// TwinCAT 3 PLC project Base_Lib
// Title: Base Library
// Company: Beckhoff UK
// Author: Chris Knight
// ProjectVersion: 3.3.0
// ProgramVersion: 3.1.4026.25
// libraries:
//   Tc2_Standard, * (Beckhoff Automation GmbH)
//   Tc2_System, * (Beckhoff Automation GmbH)
//   Tc3_EventLogger, * (Beckhoff Automation GmbH)
// project tree:
//   Base Types/Abort_Base/ I_Abortable.TcIO
//   Base Types/Cyclic_Base/ CyclicBase.TcPOU, I_Cyclic.TcIO
//   Base Types/Initialise/ I_Initialisable.TcIO
//   Base Types/Object/ I_Object.TcIO, Object.TcPOU
//   Base Types/Reset_Base/ I_Resettable.TcIO
//   Base Types/Task_Base/ I_Task.TcIO, TaskBase.TcPOU, TaskExecutionStates.TcDUT
//   Cyclic Runner/ I_HostObjects.TcIO, I_RunObjects.TcIO, ObjectRunner.TcPOU
//   Project Information/ F_GetCompany.TcPOU, F_GetTitle.TcPOU, F_GetVersion.TcPOU
//   Tracing/ AdsLogger.TcPOU, EventLogger.TcPOU, I_Trace.TcIO, I_TraceLogger.TcIO, I_TracePublisher.TcIO, TcEventSeverityExt.TcDUT, Trace.TcPOU, Tracing.TcGVL
//   Version/ Global_Version.TcGVL

// ---- Base Types/Task_Base/TaskExecutionStates.TcDUT
{attribute 'qualified_only'}
{attribute 'strict'}
{attribute 'to_string'}
TYPE TaskExecutionStates :
(
	Idle := 0,
	Running := 1,
	Done := 2,
	Error := 3
);
END_TYPE

// ---- Tracing/TcEventSeverityExt.TcDUT
{attribute 'qualified_only'}
{attribute 'strict'}
{attribute 'to_string'}
TYPE TcEventSeverityExt : (
		Verbose	 := 0,
		Info	 := 1,
		Warning	 := 2,
		Error	 := 3,
		Critical := 4,
		Off		 := 5
	);
END_TYPE

// ---- Tracing/Tracing.TcGVL
{attribute 'qualified_only'}
VAR_GLOBAL
	Trace : Trace<10> := (TraceLevel := TcEventSeverityExt.Verbose);
	{attribute 'hide'}
	AdsLogger : AdsLogger(Trace);
	TcEventLogger : EventLogger(Trace);
END_VAR

// ---- Version/Global_Version.TcGVL
{attribute 'TcGenerated'}
{attribute 'no-analysis'}
{attribute 'linkalways'}
// This function has been automatically generated from the project information.
VAR_GLOBAL CONSTANT
	{attribute 'const_non_replaced'}
	stLibVersion_Base_Library : ST_LibVersion := (iMajor := 3, iMinor := 3, iBuild := 0, iRevision := 0, nFlags := 0, sVersion := '3.3.0');
END_VAR

// ---- Base Types/Abort_Base/I_Abortable.TcIO
INTERFACE I_Abortable EXTENDS __SYSTEM.IQueryInterface

METHOD Abort : HRESULT
VAR_INPUT
END_VAR
END_METHOD

END_INTERFACE

// ---- Base Types/Cyclic_Base/I_Cyclic.TcIO
INTERFACE I_Cyclic EXTENDS __SYSTEM.IQueryInterface

METHOD PUBLIC Cycle : HRESULT
VAR_INPUT
END_VAR
END_METHOD

END_INTERFACE

// ---- Base Types/Initialise/I_Initialisable.TcIO
INTERFACE I_Initialisable EXTENDS __SYSTEM.IQueryInterface

METHOD Initialise : HRESULT
VAR_INPUT
END_VAR
END_METHOD

PROPERTY Initialised : BOOL
GET
END_GET
END_PROPERTY

END_INTERFACE

// ---- Base Types/Object/I_Object.TcIO
INTERFACE I_Object

METHOD RegisterWithParent
VAR_INPUT
	Parent : I_HostObjects;
END_VAR
END_METHOD

END_INTERFACE

// ---- Base Types/Reset_Base/I_Resettable.TcIO
INTERFACE I_Resettable

METHOD PUBLIC Reset : HRESULT
VAR_INPUT
END_VAR
END_METHOD

END_INTERFACE

// ---- Base Types/Task_Base/I_Task.TcIO
INTERFACE I_Task EXTENDS I_Cyclic

PROPERTY Busy : bool
GET
END_GET
END_PROPERTY

PROPERTY Done : bool
GET
END_GET
END_PROPERTY

PROPERTY Error : bool
GET
END_GET
END_PROPERTY

END_INTERFACE

// ---- Cyclic Runner/I_HostObjects.TcIO
INTERFACE I_HostObjects

METHOD RegisterAbortable : HRESULT
VAR_INPUT
	Abortable : I_Abortable;
END_VAR
END_METHOD

METHOD RegisterCyclic : HRESULT
VAR_INPUT
	Cyclic : I_Cyclic;
END_VAR
END_METHOD

METHOD RegisterInitialisable : HRESULT
VAR_INPUT
	Initialisable : I_Initialisable;
END_VAR
END_METHOD

METHOD RegisterObject : HRESULT
VAR_INPUT
	Object : I_Object;
END_VAR
END_METHOD

METHOD RegisterResettable : HRESULT
VAR_INPUT
	Resetable : I_Resettable;
END_VAR
END_METHOD

METHOD RegisterTask : HRESULT
VAR_INPUT
	Task : I_Task;
END_VAR
END_METHOD

END_INTERFACE

// ---- Cyclic Runner/I_RunObjects.TcIO
INTERFACE I_RunObjects

METHOD Abort : HRESULT
VAR_INPUT
END_VAR
END_METHOD

METHOD PUBLIC  Cycle : HRESULT
VAR_INPUT
END_VAR
END_METHOD

METHOD DeregisterAll : HRESULT
VAR_INPUT
END_VAR
END_METHOD

METHOD Initialise : HRESULT
END_METHOD

METHOD Initialise_Ordered : HRESULT
END_METHOD

METHOD Register : HRESULT
VAR_INPUT
	Registerable : I_Object;
END_VAR
END_METHOD

METHOD Reset : HRESULT
VAR_INPUT
END_VAR
END_METHOD

END_INTERFACE

// ---- Tracing/I_Trace.TcIO
INTERFACE I_Trace

METHOD Critical
VAR_INPUT
	Source	  : T_MaxString;
	Message	  : T_MaxString;
END_VAR
END_METHOD

METHOD Error
VAR_INPUT
	Source	  : T_MaxString;
	Message	  : T_MaxString;
END_VAR
END_METHOD

METHOD Info
VAR_INPUT
	Source	  : T_MaxString;
	Message	  : T_MaxString;
END_VAR
END_METHOD

METHOD Verbose
VAR_INPUT
	Source	  : T_MaxString;
	Message	  : T_MaxString;
END_VAR
END_METHOD

METHOD Warning
VAR_INPUT
	Source	  : T_MaxString;
	Message	  : T_MaxString;
END_VAR
END_METHOD

END_INTERFACE

// ---- Tracing/I_TraceLogger.TcIO
INTERFACE I_TraceLogger

METHOD LogMessage
VAR_INPUT
	Key		  : T_MaxString;
	Value	  : T_MaxString;
	SourceId  : UDINT := 0;
	TimeStamp : ULINT := 0;
	MessageId : UDINT := 1;
	Severity  : USINT := 1;
END_VAR
END_METHOD

END_INTERFACE

// ---- Tracing/I_TracePublisher.TcIO
INTERFACE I_TracePublisher

METHOD Subscribe
VAR_INPUT
	Logger : I_TraceLogger;
END_VAR
END_METHOD

METHOD Unsubscribe
VAR_INPUT
	Logger : I_TraceLogger;
END_VAR
END_METHOD

END_INTERFACE

// ---- Tracing/Trace.TcPOU
FUNCTION_BLOCK Trace
VAR_GENERIC CONSTANT
	MaxCount : UDINT := 10;
END_VAR IMPLEMENTS I_TracePublisher, I_Trace
VAR
	Loggers : ARRAY[0..MaxCount] OF I_TraceLogger;
	_TraceLevel : TcEventSeverityExt := TcEventSeverityExt.Warning;
END_VAR

METHOD Critical
VAR_INPUT
	Source	  : T_MaxString;
	Message	  : T_MaxString;
END_VAR
VAR
	i : UDINT;
END_VAR
FOR i := 0 TO MaxCount DO
	IF Loggers[i] <> 0 AND_THEN _TraceLevel < 5 THEN
		Loggers[i].LogMessage(Source,
							  Message,
							  0,
							  0,
							  1,
							  4);
	END_IF
END_FOR
END_METHOD

METHOD Error
VAR_INPUT
	Source	  : T_MaxString;
	Message	  : T_MaxString;
END_VAR
VAR
	i : UDINT;
END_VAR
FOR i := 0 TO MaxCount DO
	IF Loggers[i] <> 0 AND_THEN _TraceLevel < 4 THEN
		Loggers[i].LogMessage(Source,
							  Message,
							  0,
							  0,
							  1,
							  3);
	END_IF
END_FOR
END_METHOD

METHOD Info
VAR_INPUT
	Source	  : T_MaxString;
	Message	  : T_MaxString;
END_VAR
VAR
	i : UDINT;
END_VAR
FOR i := 0 TO MaxCount DO
	IF Loggers[i] <> 0 AND_THEN _TraceLevel < 2 THEN
		Loggers[i].LogMessage(Source,
							  Message,
							  0,
							  0,
							  1,
							  1);
	END_IF
END_FOR
END_METHOD

METHOD Subscribe
VAR_INPUT
	Logger : I_TraceLogger;
END_VAR

VAR
	i : UDINT;
END_VAR
FOR i := 0 TO MaxCount DO
	IF Loggers[i] = 0 THEN
		Loggers[i] := Logger;
		EXIT;
	END_IF
END_FOR
END_METHOD

PROPERTY TraceLevel : TcEventSeverityExt
GET
TraceLevel := _TraceLevel;
END_GET
SET
_TraceLevel := TraceLevel;
END_SET
END_PROPERTY

METHOD Unsubscribe
VAR_INPUT
	Logger : I_TraceLogger;
END_VAR

VAR
	i : UDINT;
END_VAR
FOR i := 0 TO MaxCount DO
	IF Loggers[i] = Logger THEN
		Loggers[i] := 0;
		EXIT;
	END_IF
END_FOR
END_METHOD

METHOD Verbose
VAR_INPUT
	Source	  : T_MaxString;
	Message	  : T_MaxString;
END_VAR
VAR
	i : UDINT;
END_VAR
FOR i := 0 TO MaxCount DO
	IF Loggers[i] <> 0 AND_THEN _TraceLevel = 0 THEN
		Loggers[i].LogMessage(Source,
							  Message,
							  0,
							  0,
							  1,
							  0);
	END_IF
END_FOR
END_METHOD

METHOD Warning
VAR_INPUT
	Source	  : T_MaxString;
	Message	  : T_MaxString;
END_VAR
VAR
	i : UDINT;
END_VAR
FOR i := 0 TO MaxCount DO
	IF Loggers[i] <> 0 AND_THEN _TraceLevel < 3 THEN
		Loggers[i].LogMessage(Source,
							  Message,
							  0,
							  0,
							  1,
							  2);
	END_IF
END_FOR
END_METHOD

END_FUNCTION_BLOCK

// ---- Tracing/AdsLogger.TcPOU
FUNCTION_BLOCK AdsLogger IMPLEMENTS I_TraceLogger
VAR
	MessagesThisScan : DINT;
	CurrentCycle	 : UDINT;
END_VAR

//FB_Init is always available implicitly and it is used primarily for initialization.

//The return value is not evaluated. For a specific influence, you can also declare the

//methods explicitly and provide additional code there with the standard initialization

//code. You can evaluate the return value.
METHOD FB_Init : BOOL
VAR_INPUT
	bInitRetains   : BOOL; // TRUE: the retain variables are initialized (reset warm / reset cold)
	bInCopyCode	   : BOOL; // TRUE: the instance will be copied to the copy code afterward (online change)   
	TracePublisher : I_TracePublisher;
END_VAR
TracePublisher.Subscribe(THIS^);
END_METHOD

METHOD LogMessage
VAR_INPUT
	Key		  : T_MaxString;
	Value	  : T_MaxString;
	SourceId  : UDINT := 0;
	TimeStamp : ULINT := 0;
	MessageId : UDINT := 1;
	Severity  : USINT := 1;
END_VAR
IF TwinCAT_SystemInfoVarList._TaskInfo[GETCURTASKINDEXEX()].CycleCount <> CurrentCycle THEN
	CurrentCycle	 := TwinCAT_SystemInfoVarList._TaskInfo[GETCURTASKINDEXEX()].CycleCount;
	MessagesThisScan := 0;
END_IF

IF NOT (MessagesThisScan < TO_DINT(TwinCAT_SystemInfoVarList._TaskInfo[GETCURTASKINDEXEX()].CycleTime / 2000)) THEN
	RETURN;
END_IF

IF MessagesThisScan < TO_DINT(TwinCAT_SystemInfoVarList._TaskInfo[GETCURTASKINDEXEX()].CycleTime / 2000) THEN
	CASE Severity OF
		0,1:
			ADSLOGSTR(ADSLOG_MSGTYPE_LOG OR ADSLOG_MSGTYPE_HINT, Concat(Key, ': %s'), Value);
		2:
			ADSLOGSTR(ADSLOG_MSGTYPE_LOG OR ADSLOG_MSGTYPE_WARN, Concat(Key, ': %s'), Value);
		3,4:
			ADSLOGSTR(ADSLOG_MSGTYPE_LOG OR ADSLOG_MSGTYPE_ERROR, Concat(Key, ': %s'), Value);
	END_CASE
	
	MessagesThisScan := MessagesThisScan + 1;
END_IF
END_METHOD

END_FUNCTION_BLOCK

// ---- Tracing/EventLogger.TcPOU
FUNCTION_BLOCK EventLogger IMPLEMENTS I_TraceLogger
VAR
	MessagesThisScan : DINT;
	Message			 : FB_TcMessage;
	Source			 : FB_TcSourceInfo;
	CurrentCycle	 : UDINT;
END_VAR

//FB_Init is always available implicitly and it is used primarily for initialization.
//The return value is not evaluated. For a specific influence, you can also declare the
//methods explicitly and provide additional code there with the standard initialization
//code. You can evaluate the return value.
METHOD FB_Init: BOOL
VAR_INPUT
    bInitRetains: BOOL; // TRUE: the retain variables are initialized (reset warm / reset cold)
    bInCopyCode: BOOL;  // TRUE: the instance will be copied to the copy code afterward (online change)   
	TracePublisher : I_TracePublisher;	
END_VAR
TracePublisher.Subscribe(THIS^);
END_METHOD

METHOD LogMessage
VAR_INPUT
	Key	: T_MaxString;
	Value	: T_MaxString;
	SourceId	: UDINT := 0;
	TimeStamp	: ULINT := 0;
	MessageId	: UDINT := 1;
	Severity	: USINT := 1;
END_VAR
VAR
	EventSeverity : TcEventSeverity;
END_VAR
IF TwinCAT_SystemInfoVarList._TaskInfo[GETCURTASKINDEXEX()].CycleCount <> CurrentCycle THEN
	CurrentCycle	 := TwinCAT_SystemInfoVarList._TaskInfo[GETCURTASKINDEXEX()].CycleCount;
	MessagesThisScan := 0;
END_IF

IF NOT (MessagesThisScan < TO_DINT(TwinCAT_SystemInfoVarList._TaskInfo[GETCURTASKINDEXEX()].CycleTime / 2000)) THEN
	RETURN;
END_IF

CASE Severity OF
	0: 
		EventSeverity := TcEventSeverity.Verbose;

	1:
		EventSeverity := TcEventSeverity.Info;

	2:
		EventSeverity := TcEventSeverity.Warning;

	3:
		EventSeverity := TcEventSeverity.Error;

	4:
		EventSeverity := TcEventSeverity.Critical;
END_CASE

Source.sName := Key;
Source.nId	 := SourceId;
Message.Create(eventClass	:= TC_EVENT_CLASSES.TraceEvents,
			   nEventId		:= MessageId,
			   eSeverity	:= EventSeverity,
			   ipSourceInfo := Source);

Message.ipArguments.Clear().AddString(Value);
Message.Send(TimeStamp);
Message.Release();
Source.Clear();
MessagesThisScan := MessagesThisScan + 1;
END_METHOD

END_FUNCTION_BLOCK

// ---- Base Types/Cyclic_Base/CyclicBase.TcPOU
FUNCTION_BLOCK ABSTRACT CyclicBase EXTENDS Object IMPLEMENTS I_Cyclic
VAR
END_VAR

{analysis -2}

METHOD PUBLIC ABSTRACT Cycle : HRESULT
VAR_INPUT
END_VAR
{analysis -2}
END_METHOD

METHOD RegisterWithParent
VAR_INPUT
	Parent	: I_HostObjects;
END_VAR
Parent.RegisterObject(THIS^);
Parent.RegisterCyclic(THIS^);
END_METHOD

END_FUNCTION_BLOCK

// ---- Base Types/Object/Object.TcPOU
FUNCTION_BLOCK ABSTRACT Object IMPLEMENTS I_Object
VAR
	_Name : T_MaxString;
END_VAR

//FB_Init is always available implicitly and it is used primarily for initialization.
//The return value is not evaluated. For a specific influence, you can also declare the
//methods explicitly and provide additional code there with the standard initialization
//code. You can evaluate the return value.
METHOD FB_Init: BOOL
VAR_INPUT
    bInitRetains: BOOL; // TRUE: the retain variables are initialized (reset warm / reset cold)
    bInCopyCode: BOOL;  // TRUE: the instance will be copied to the copy code afterward (online change)  
	Name : T_MaxString; 
END_VAR
_Name := Name;
END_METHOD

PROPERTY Name : T_MaxString
GET
Name := _Name;
END_GET
END_PROPERTY

METHOD RegisterWithParent
VAR_INPUT
	Parent	: I_HostObjects;
END_VAR
Parent.RegisterObject(THIS^);
END_METHOD

END_FUNCTION_BLOCK

// ---- Base Types/Task_Base/TaskBase.TcPOU
FUNCTION_BLOCK ABSTRACT TaskBase EXTENDS CyclicBase IMPLEMENTS I_Task
VAR
	_Busy : BOOL;
	_Error : BOOL;
	_Done : BOOL;
	State: INT;
END_VAR

{analysis -2}

PROPERTY Busy : BOOL
GET
Busy := _Busy;
END_GET
END_PROPERTY

PROPERTY Done : BOOL
GET
Done := _Done;
END_GET
END_PROPERTY

PROPERTY Error : BOOL
GET
Error := _Error;
END_GET
END_PROPERTY

END_FUNCTION_BLOCK

// ---- Cyclic Runner/ObjectRunner.TcPOU
FUNCTION_BLOCK ObjectRunner 
VAR_GENERIC CONSTANT
	MaxRegisteredModules : INT := 99;
END_VAR IMPLEMENTS I_Cyclic, I_HostObjects, I_RunObjects
VAR
	Objects : ARRAY[0..MaxRegisteredModules] OF I_Object;
	CyclicModules : ARRAY[0..MaxRegisteredModules] OF I_Cyclic;
	InitialiseModules : ARRAY[0..MaxRegisteredModules] OF I_Initialisable;
	ResetableModules : ARRAY[0..MaxRegisteredModules] OF I_Resettable;
	AbortableModules : ARRAY[0..MaxRegisteredModules] OF I_Abortable;
	TaskModules : ARRAY[0..MaxRegisteredModules] OF I_Task;
	_ObjectCount : INT := 0;
	_CyclicModuleCount : INT := 0;
	_InitModuleCount : INT := 0;
	_ResetModuleCount : INT := 0;
	_TaskModuleCount : INT := 0;
	_AbortModuleCount: INT := 0;
	InitialisationCount : INT := 0;
	Registered: BOOL;
	_AllInitialised : BOOL := TRUE;
END_VAR

METHOD Abort : HRESULT
VAR_INPUT
END_VAR
VAR	
	i: INT;
END_VAR
IF _AbortModuleCount = 0 THEN
	Abort := -1;
	RETURN;
END_IF

FOR i := 0 TO _AbortModuleCount - 1 DO
	IF AbortableModules[i] <> 0 THEN
		AbortableModules[i].Abort();
	END_IF
END_FOR
END_METHOD

PROPERTY AbortableModuleCount : INT
GET
AbortableModuleCount := _AbortModuleCount;
END_GET
END_PROPERTY

METHOD PUBLIC  Cycle : HRESULT
VAR_INPUT
END_VAR
VAR	
	i: INT;
END_VAR
FOR i := 0 TO _CyclicModuleCount -1 DO
	IF CyclicModules[i] <> 0 THEN
		CyclicModules[i].Cycle();
	END_IF
END_FOR
END_METHOD

PROPERTY CyclicModuleCount : INT
GET
CyclicModuleCount := _CyclicModuleCount;
END_GET
END_PROPERTY

METHOD DeregisterAll : HRESULT
VAR_INPUT
END_VAR
VAR	
	i: INT;
END_VAR
FOR i := 0 TO MaxRegisteredModules DO
	Objects[i] := 0;
	CyclicModules[i] := 0;
	InitialiseModules[i] := 0;
	ResetableModules[i] := 0;
	AbortableModules[i] := 0;
	TaskModules[i] := 0;
END_FOR
_CyclicModuleCount := 0;
_InitModuleCount := 0;
_ResetModuleCount := 0;
_TaskModuleCount := 0;
_AbortModuleCount := 0;
InitialisationCount := 0;
_ObjectCount := 0;
DeregisterAll := 1;
END_METHOD

PROPERTY InitialisableModuleCount : INT
GET
InitialisableModuleCount := _InitModuleCount;
END_GET
END_PROPERTY

PROPERTY InitialisationComplete : BOOL
GET
InitialisationComplete := _AllInitialised;
END_GET
END_PROPERTY

METHOD Initialise : HRESULT
VAR
	i : INT;
END_VAR
IF _InitModuleCount = 0 THEN
	_AllInitialised := TRUE;
	RETURN; 
END_IF

_AllInitialised := TRUE;
FOR i := 0 TO _InitModuleCount DO
	IF InitialiseModules[i] <> 0 THEN 
		IF NOT InitialiseModules[i].Initialised THEN
			InitialiseModules[i].Initialise();
			_AllInitialised := FALSE;
			Initialise := -1;
		END_IF
	END_IF
END_FOR
END_METHOD

METHOD Initialise_Ordered : HRESULT
VAR
	i : INT;
END_VAR
IF _InitModuleCount = 0 THEN
	_AllInitialised := TRUE;
	RETURN; 
END_IF

IF InitialisationCount < MaxRegisteredModules THEN
	IF InitialiseModules[InitialisationCount] <> 0 THEN
		IF NOT InitialiseModules[InitialisationCount].Initialised THEN
			InitialiseModules[InitialisationCount].Initialise();
		ELSE
			InitialisationCount := InitialisationCount + 1;
		END_IF
		Initialise_Ordered := -1;
	ELSE
		InitialisationCount := InitialisationCount + 1;
	END_IF
ELSE
	InitialisationCount := 0;
	_AllInitialised := TRUE;
END_IF
END_METHOD

METHOD Register : HRESULT
VAR_INPUT
	Registerable : I_Object;
END_VAR
IF Registerable = 0 THEN
	Register := -1;
	RETURN;
END_IF

Registerable.RegisterWithParent(THIS^);
END_METHOD

METHOD RegisterAbortable : HRESULT
VAR_INPUT
	Abortable : I_Abortable;
END_VAR
VAR	
	i: INT;
END_VAR
IF Abortable = 0 THEN
	RegisterAbortable := -1;
	RETURN;
END_IF

IF _AbortModuleCount >= MaxRegisteredModules THEN
	RegisterAbortable := -2;
	RETURN;
END_IF

Registered := FALSE;
FOR i := 0 TO MaxRegisteredModules DO
	IF AbortableModules[i] = Abortable THEN
		Registered := TRUE;
	END_IF
END_FOR

IF Registered THEN
	RegisterAbortable := -3;
	RETURN;
END_IF

FOR i := 0 TO MaxRegisteredModules DO
	IF AbortableModules[i] = 0 THEN
		AbortableModules[i] := Abortable;
		_AbortModuleCount := _AbortModuleCount + 1;
		EXIT;
	END_IF
END_FOR
END_METHOD

METHOD RegisterCyclic : HRESULT
VAR_INPUT
	Cyclic : I_Cyclic;
END_VAR
VAR	
	i: INT;
END_VAR
IF Cyclic = 0 THEN
	RegisterCyclic := -1;
	RETURN;
END_IF

IF _CyclicModuleCount >= MaxRegisteredModules THEN
	RegisterCyclic := -2;
	RETURN;
END_IF

Registered := FALSE;
FOR i := 0 TO MaxRegisteredModules DO
	IF CyclicModules[i] = Cyclic THEN
		Registered := TRUE;
	END_IF
END_FOR

IF Registered THEN
	RegisterCyclic := -3;
	RETURN;
END_IF

FOR i := 0 TO MaxRegisteredModules DO
	IF CyclicModules[i] = 0 THEN
		CyclicModules[i] := Cyclic;
		_CyclicModuleCount := _CyclicModuleCount + 1;
		EXIT;
	END_IF
END_FOR
END_METHOD

PROPERTY RegisteredObjectCount : INT
GET
RegisteredObjectCount := _ObjectCount;
END_GET
END_PROPERTY

METHOD RegisterInitialisable : hresult
VAR_INPUT
	Initialisable : I_Initialisable;
END_VAR
VAR	
	i: INT;
END_VAR
IF Initialisable = 0 THEN
	RegisterInitialisable := -1;
	RETURN;
END_IF

IF _InitModuleCount >= MaxRegisteredModules THEN
	RegisterInitialisable := -2;
	RETURN;
END_IF

Registered := FALSE;
FOR i := 0 TO MaxRegisteredModules DO
	IF InitialiseModules[i] = Initialisable THEN
		Registered := TRUE;
	END_IF
END_FOR

IF Registered THEN
	RegisterInitialisable := -3;
	RETURN;
END_IF

FOR i := 0 TO MaxRegisteredModules DO
	IF InitialiseModules[i] = 0 THEN
		InitialiseModules[i] := Initialisable;
		_InitModuleCount := _InitModuleCount + 1;
		EXIT;
	END_IF
END_FOR
END_METHOD

METHOD RegisterObject : HRESULT
VAR_INPUT
	Object : I_Object;
END_VAR
VAR	
	i: INT;
END_VAR
IF Object = 0 THEN
	RegisterObject := -1;
	RETURN;
END_IF

IF _ObjectCount >= MaxRegisteredModules THEN
	RegisterObject := -2;
	RETURN;
END_IF

Registered := FALSE;
FOR i := 0 TO MaxRegisteredModules DO
	IF Objects[i] = Object THEN
		Registered := TRUE;
	END_IF
END_FOR

IF Registered THEN
	RegisterObject := -3;
	RETURN;
END_IF

FOR i := 0 TO MaxRegisteredModules DO
	IF Objects[i] = 0 THEN
		Objects[i] := Object;
		_ObjectCount := _ObjectCount + 1;
		EXIT;
	END_IF
END_FOR
END_METHOD

METHOD RegisterResettable : HRESULT
VAR_INPUT
	Resetable : I_Resettable;
END_VAR
VAR	
	i: INT;
END_VAR
IF Resetable = 0 THEN
	RegisterResettable := -1;
	RETURN;
END_IF

IF _ResetModuleCount >= MaxRegisteredModules THEN
	RegisterResettable := -2;
	RETURN;
END_IF

Registered := FALSE;
FOR i := 0 TO MaxRegisteredModules DO
	IF ResetableModules[i] = Resetable THEN
		Registered := TRUE;
	END_IF
END_FOR

IF Registered THEN
	RegisterResettable := -3;
	RETURN;
END_IF

FOR i := 0 TO MaxRegisteredModules DO
	IF ResetableModules[i] = 0 THEN
		ResetableModules[i] := Resetable;
		_ResetModuleCount := _ResetModuleCount + 1;
		EXIT;
	END_IF
END_FOR
END_METHOD

METHOD RegisterTask : HRESULT
VAR_INPUT
	Task : I_Task;
END_VAR
VAR	
	i: INT;
END_VAR
IF Task = 0 THEN
	RegisterTask := -1;
	RETURN;
END_IF

IF _TaskModuleCount >= MaxRegisteredModules THEN
	RegisterTask := -2;
	RETURN;
END_IF

Registered := FALSE;
FOR i := 0 TO MaxRegisteredModules DO
	IF TaskModules[i] = Task THEN
		Registered := TRUE;
	END_IF
END_FOR

IF Registered THEN
	RegisterTask := -3;
	RETURN;
END_IF

FOR i := 0 TO MaxRegisteredModules DO
	IF TaskModules[i] = 0 THEN
		TaskModules[i] := Task;
		_TaskModuleCount := _TaskModuleCount + 1;
		EXIT;
	END_IF
END_FOR
END_METHOD

METHOD Reset : HRESULT
VAR_INPUT
END_VAR
VAR	
	i: INT;
END_VAR
FOR i := 0 TO _ResetModuleCount - 1 DO
	IF ResetableModules[i] <> 0 THEN
		ResetableModules[i].Reset();
	END_IF
END_FOR
END_METHOD

PROPERTY ResettableModuleCount : INT
GET
ResettableModuleCount := _ResetModuleCount;
END_GET
END_PROPERTY

PROPERTY TaskModuleCount : INT
GET
TaskModuleCount := _TaskModuleCount;
END_GET
END_PROPERTY

END_FUNCTION_BLOCK

// ---- Project Information/F_GetCompany.TcPOU
// This function has been automatically generated from the project information.
{attribute 'signature_flag' := '1073741824'}
{attribute 'TcGenerated'}
{attribute 'no-analysis'}
FUNCTION F_GetCompany : WSTRING
VAR_INPUT
	
END_VAR

F_GetCompany := "Beckhoff UK";

END_FUNCTION

// ---- Project Information/F_GetTitle.TcPOU
// This function has been automatically generated from the project information.
{attribute 'signature_flag' := '1073741824'}
{attribute 'TcGenerated'}
{attribute 'no-analysis'}
FUNCTION F_GetTitle : WSTRING
VAR_INPUT
	
END_VAR

F_GetTitle := "Base Library";

END_FUNCTION

// ---- Project Information/F_GetVersion.TcPOU
// This function has been automatically generated from the project information.
{attribute 'signature_flag' := '1073741824'}
{attribute 'TcGenerated'}
{attribute 'no-analysis'}
FUNCTION F_GetVersion : ST_LibVersion
VAR_INPUT
	
END_VAR

F_GetVersion.iMajor := 3;
F_GetVersion.iMinor := 3;
F_GetVersion.iBuild := 0;
F_GetVersion.iRevision := 0;
F_GetVersion.sVersion := '3.3.0';
F_GetVersion.nFlags := 0;

END_FUNCTION
